Staubli VAL3: GetPreset.pgx

public program GetPreset(num& x_nPreset[] (dimensions=1), num x_nPrecent (dimensions=1), num x_nPWMH (dimensions=1), num x_nPWML (dimensions=1))
  local num l_nNum
  local num l_nPWM
begin

  x_nPreset[0]=aioGet(aAio["O1_aLasPwr"])
  x_nPreset[1]=aioGet(aAio["O1_aFPWM"])
  x_nPreset[2]=aioGet(aAio["O1_aPMW"])
  x_nPreset[3]=aioGet(aAio["O1_aAirPress"])
  x_nPreset[4]=aioGet(aAio["O2_aFollowSensitive"])

  for l_nNum=0 to 4
    if l_nNum==1
      //强制设置为1500
      l_nPWM=x_nPWMH-x_nPWML
      l_nPWM=sel(l_nPWM<1,1,l_nPWM)
      x_nPreset[1]=(x_nPreset[1]-x_nPWML)/l_nPWM*100
    else
      if l_nNum!=2
        x_nPreset[l_nNum]=round(x_nPreset[l_nNum]/max(x_nPrecent,1)*100)
      endIf
    endIf
  endFor



end
